FUNCTION_BLOCK CMD_bloc_FV
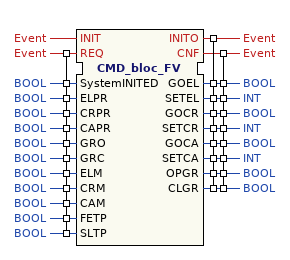
  EVENT_INPUT
    INIT;
    REQ WITH SystemINITED, ELPR, CRPR, CAPR, GRO, GRC, ELM, CRM, CAM, FETP, SLTP;
  END_EVENT
  EVENT_OUTPUT
    INITO WITH GOEL, SETEL, GOCA, SETCA, GOCR, SETCR, OPGR, CLGR;
    CNF WITH GOEL, SETEL, GOCA, SETCA, GOCR, SETCR, OPGR, CLGR;
  END_EVENT
  VAR_INPUT
    SystemINITED : BOOL;
    ELPR : BOOL;
    CRPR : BOOL;
    CAPR : BOOL;
    GRO : BOOL;
    GRC : BOOL;
    ELM : BOOL;
    CRM : BOOL;
    CAM : BOOL;
    FETP : BOOL;
    SLTP : BOOL;
  END_VAR
  VAR_OUTPUT
    GOEL : BOOL;
    SETEL : INT;
    GOCR : BOOL;
    SETCR : INT;
    GOCA : BOOL;
    SETCA : INT;
    OPGR : BOOL;
    CLGR : BOOL;
  END_VAR
  EC_STATES
    START;
    INIT : INIT -> INITO;
    CR_01_CA_03 : GOCA_06 -> CNF;
    CR_01_03_CA_06 : GOCR_03 -> CNF;
    GRC_03_GRC_04 : GOCR_01 -> CNF;
    CR_01_CA_06_f : GO_CA_CR_EL -> CNF;
    EL_03 : OPGR -> CNF;
    GRO : GOCR_01 -> CNF;
    EL_01 : GOCR_01 -> CNF;
    CR_01_EL_03 : GOCA_01 -> CNF;
    CR_01_CA_01_e : GOCR_02 -> CNF;
    CR_02_CA_01 : CLGR -> CNF;
    GRC : GOCR_01 -> CNF;
    CR_01_CA_01_f : GOCA_03 -> CNF;
    CR_01_CA_03_lid : GOCR_03 -> CNF;
    CR_03_CA_03 : OPGR -> CNF;
    GRO_lid : GOEL_01 -> CNF;
    CR_01_EL_01 : RESET -> CNF;
    CR_01_CA_06_e : RESET -> CNF;
    CR_03_CA_06 : CLGR -> CNF;
    CR_01_04_CA_06 : GOCR_04 -> CNF;
    CR_04_CA_06 : CLGR -> CNF;
    ReadyToDrop : STOP_CR -> CNF;
  END_STATES
  EC_TRANSITIONS
    START TO INIT := INIT;
    CR_01_03_CA_06 TO CR_03_CA_06 := [NOT CRM & CRPR];
    GRC_03_GRC_04 TO ReadyToDrop := [NOT CRM & CRPR];
    EL_03 TO GRO := GRO;
    GRO TO CR_01_EL_03 := [NOT CRM & CRPR];
    CR_01_EL_03 TO CR_01_CA_01_e := [NOT CAM & CAPR];
    CR_01_CA_01_e TO CR_02_CA_01 := [NOT CRM & CRPR];
    CR_02_CA_01 TO GRC := GRC;
    GRC TO CR_01_CA_01_f := [NOT CRM & CRPR];
    CR_01_CA_01_f TO CR_01_CA_03_lid := [NOT CAM & CAPR];
    CR_01_CA_03_lid TO CR_03_CA_03 := [NOT CRM & CRPR];
    CR_03_CA_03 TO GRO_lid := GRO;
    GRO_lid TO EL_01 := [NOT ELM & ELPR];
    EL_01 TO CR_01_EL_01 := [NOT CRM & CRPR];
    CR_01_CA_03 TO CR_01_CA_06_e := [NOT CAM & CAPR];
    CR_01_CA_06_e TO CR_01_03_CA_06 := FETP;
    CR_03_CA_06 TO GRC_03_GRC_04 := GRC;
    INIT TO CR_01_CA_03 := [SystemINITED & (FETP OR SLTP)];
    CR_01_EL_01 TO CR_01_CA_03 := 1;
    CR_01_04_CA_06 TO CR_04_CA_06 := [NOT CRM & CRPR];
    CR_01_CA_06_e TO CR_01_04_CA_06 := SLTP;
    CR_04_CA_06 TO GRC_03_GRC_04 := GRC;
    CR_01_CA_06_f TO EL_03 := [(NOT CRM & CRPR) AND (NOT ELM & ELPR) AND (NOT CAM & CAPR)];
    ReadyToDrop TO CR_01_CA_06_f := REQ;
  END_TRANSITIONS
  ALGORITHM INIT IN ST:

  END_ALGORITHM
  ALGORITHM GOCA_06 IN ST:
GOCA := TRUE;
SETCA := 3;
GOEL := FALSE;
GOCR := FALSE;
  END_ALGORITHM
  ALGORITHM GOCR_03 IN ST:
GOCR := TRUE;
SETCR := 3;
GOCA := FALSE;
GOEL := FALSE;
  END_ALGORITHM
  ALGORITHM GOCR_04 IN ST:
GOCR := TRUE;
SETCR := 3;
GOEL := FALSE;
GOCA := FALSE;
  END_ALGORITHM
  ALGORITHM CLGR IN ST:
CLGR := TRUE;
OPGR := FALSE;
GOCR := FALSE;
GOEL := FALSE;
GOCA := FALSE;
  END_ALGORITHM
  ALGORITHM GOCR_01 IN ST:
GOCR := TRUE;
SETCR := 1;
GOCA := FALSE;
GOEL := FALSE;
FETP := FALSE;
SLTP := FALSE;
  END_ALGORITHM
  ALGORITHM GOCA_03 IN ST:
GOCA := TRUE;
SETCA := 2;
GOEL := FALSE;
GOCR := FALSE;
  END_ALGORITHM
  ALGORITHM GOCR_06 IN ST:
GOCR := TRUE;
SETCR := 4;
GOCA := FALSE;
GOEL := FALSE;
  END_ALGORITHM
  ALGORITHM GOEL_03 IN ST:
GOEL := TRUE;
SETEL := 2;
GOCA := FALSE;
GOCR := FALSE;
  END_ALGORITHM
  ALGORITHM OPGR IN ST:
CLGR := FALSE;
OPGR := TRUE;
GOCR := FALSE;
GOEL := FALSE;
GOCA := FALSE;
  END_ALGORITHM
  ALGORITHM GOCA_01 IN ST:
GOCA := TRUE;
SETCA := 1;
GOEL := FALSE;
GOCR := FALSE;
  END_ALGORITHM
  ALGORITHM GOCR_02 IN ST:
GOCR := TRUE;
SETCR := 2;
GOCA := FALSE;
GOEL := FALSE;
  END_ALGORITHM
  ALGORITHM GOEL_01 IN ST:
GOEL := TRUE;
SETEL := 1;
GOCA := FALSE;
GOCR := FALSE;
  END_ALGORITHM
  ALGORITHM RESET IN ST:
GOCA := FALSE;
GOCR := FALSE;
GOEL := FALSE;
OPGR := FALSE;
CLGR := FALSE;
  END_ALGORITHM
  ALGORITHM STOP IN ST:
GOCA := FALSE;
GOCR := FALSE;
GOEL := FALSE;
OPGR := FALSE;
CLGR := FALSE;
  END_ALGORITHM
  ALGORITHM GO_CA_CR_EL IN ST:
GOCA := TRUE;
SETCA := 2;
GOCR := TRUE;
SETCR := 4;
GOEL := TRUE;
SETEL := 2;
  END_ALGORITHM
  ALGORITHM STOP_CR IN ST:
GOCR := FALSE;
  END_ALGORITHM
END_FUNCTION_BLOCK
